// TIA Portal V18 export
VAR_GLOBAL   // PLC tag table "Analog_Clock"
   "Rotunda Angle input" AT %IW160 : Int;
   "Drive Angle input" AT %IW164 : Int;
   "Cabin Angle input" AT %IW166 : Int;
   "WireDraw Encoder input" AT %IW176 : Int;
   "Laser input" AT %IW162 : Int;
   "Left Driver Analog input" AT %QW160 : Int;
   "Right Driver Analog input" AT %QW162 : Int;
   "Cab Driver Analog input" AT %QW176 : Int;
   "Slow Mode input" AT %M226.1 : Bool;
   "Canopy Touch Memo" AT %M217.4 : Bool;
END_VAR
